FUNCTION TryConvert_UDINT_TO_DINT : BOOL
VAR_INPUT
	in : UDINT;
	out : REFERENCE TO DINT;
END_VAR

IF in > DatatypeLimits.MAX_VALUE_OF_UDINT_WHICH_CAN_BE_HELD_IN_A_DINT THEN
	RETURN;
END_IF

out := UDINT_TO_DINT(in);
TryConvert_UDINT_TO_DINT := TRUE;

END_FUNCTION

(* stored: Version 1.1.0.1, ProductVersion 3.1.4024.12
   POU TryConvert_UDINT_TO_DINT: Id {603c4095-2ae7-4994-a2f9-0acc1bb3433b}, SpecialFunc None *)
